FUNCTION_BLOCK basicValveControlOnOff (* Basic Function Block Type *)
  (* Standard: 61499-2 *)
  (* Version 0.0, 1/26/2026, Schneider Electric, Template *)
  PACKAGE Hidryco.HidrycoLib;
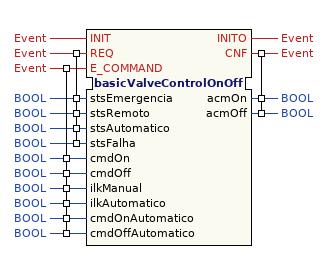
  EVENT_INPUT
    INIT; (* Initialization Request *)
    REQ WITH stsRemoto, stsAutomatico, stsFalha, stsEmergencia; (* Normal Execution Request *)
    E_COMMAND WITH cmdOn, cmdOff, ilkManual, ilkAutomatico, cmdOnAutomatico, cmdOffAutomatico;
  END_EVENT
  EVENT_OUTPUT
    INITO; (* Initialization Confirm *)
    CNF WITH acmOn, acmOff; (* Execution Confirmation *)
  END_EVENT
  VAR_INPUT
    stsEmergencia : BOOL;
    stsRemoto : BOOL;
    stsAutomatico : BOOL;
    stsFalha : BOOL;
    cmdOn : BOOL;
    cmdOff : BOOL;
    ilkManual : BOOL; (* Interlock Manual *)
    ilkAutomatico : BOOL; (* Interlock Automatico *)
    cmdOnAutomatico : BOOL;
    cmdOffAutomatico : BOOL;
  END_VAR
  VAR_OUTPUT
    acmOn : BOOL;
    acmOff : BOOL;
  END_VAR
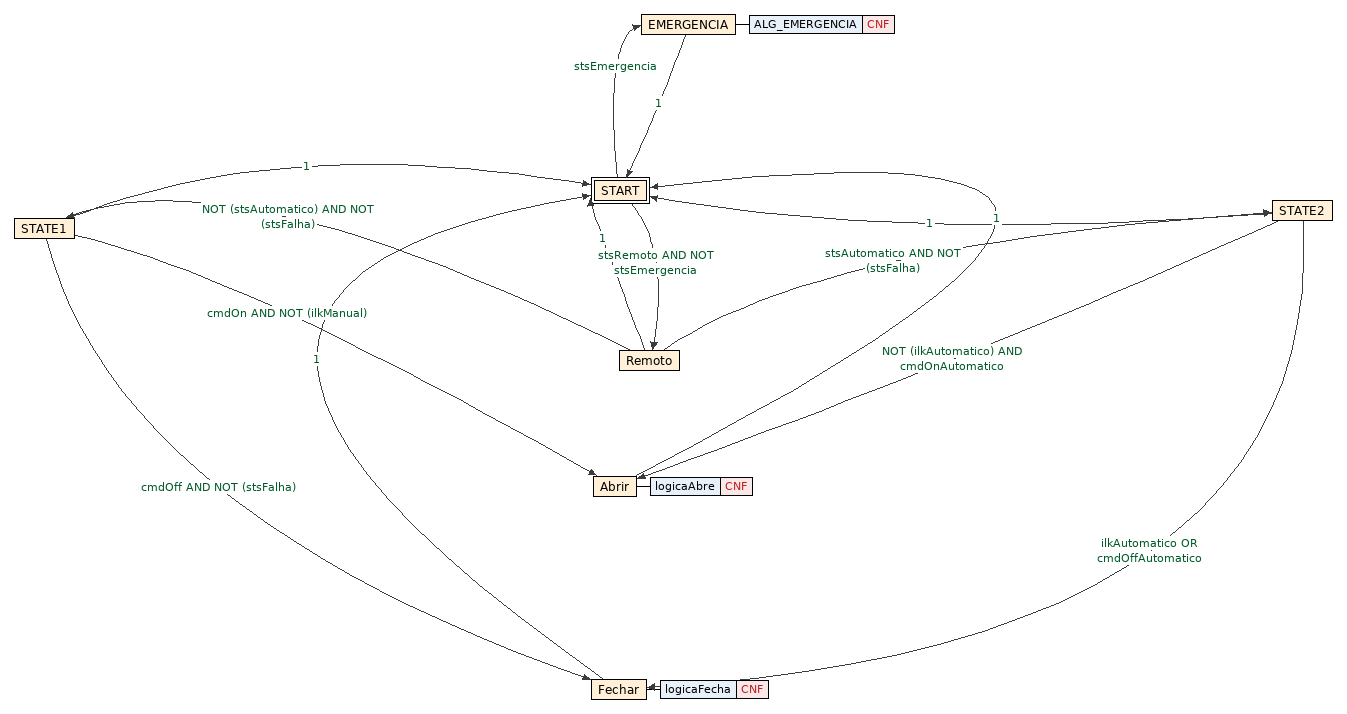
  EC_STATES
    START; (* Initial State *)
    Remoto;
    STATE2;
    STATE1;
    Abrir : logicaAbre -> CNF;
    Fechar : logicaFecha -> CNF;
    EMERGENCIA : ALG_EMERGENCIA -> CNF;
  END_STATES
  EC_TRANSITIONS
    START TO Remoto := stsRemoto AND NOT stsEmergencia;
    Remoto TO STATE2 := stsAutomatico AND NOT (stsFalha);
    Remoto TO STATE1 := NOT (stsAutomatico) AND NOT (stsFalha);
    STATE1 TO Abrir := cmdOn AND NOT (ilkManual);
    STATE1 TO Fechar := cmdOff AND NOT (stsFalha);
    STATE2 TO Abrir := NOT (ilkAutomatico) AND cmdOnAutomatico;
    STATE2 TO Fechar := ilkAutomatico OR cmdOffAutomatico;
    Remoto TO START := 1;
    Abrir TO START := 1;
    Fechar TO START := 1;
    STATE1 TO START := 1;
    STATE2 TO START := 1;
    START TO EMERGENCIA := stsEmergencia;
    EMERGENCIA TO START := 1;
  END_TRANSITIONS
  ALGORITHM INIT IN ST: (* Initialization algorithm *)
;
  END_ALGORITHM
  ALGORITHM REQ IN ST: (* Normally executed algorithm *)
;
  END_ALGORITHM
  ALGORITHM logicaFecha IN ST:
acmOn := FALSE;
acmOff := TRUE;
;
  END_ALGORITHM
  ALGORITHM logicaAbre IN ST:
acmOff := FALSE;
acmOn := TRUE;
;
  END_ALGORITHM
  ALGORITHM ALG_EMERGENCIA IN ST:
acmOff := FALSE;
acmOn := FALSE;
;
  END_ALGORITHM
END_FUNCTION_BLOCK
